(* CoDeSys 2.3.9.48 project: PLC128.pro *)
(* Libraries: WagoLibSockets.lib 14.5.12 12:49:54, SysLibSockets.lib 5.5.11 09:22:24, Standard.lib 8.11.10 12:37:48, SYSLIBCALLBACK.LIB 8.11.10 12:37:48, NETVARUDP_LIB_V23.LIB 8.11.10 12:37:48 *)

(* PLC configuration (modules and I/O channels)
IN1 AT %IX2.0 [BOOLOnX_I] Ch_1 Digital input
IN2 AT %IX2.1 [BOOLOnX_I] Ch_2 Digital input
IN3 AT %IX2.2 [BOOLOnX_I] Ch_3 Digital input
IN4 AT %IX2.3 [BOOLOnX_I] Ch_4 Digital input
IN5 AT %IX2.4 [BOOLOnX_I] Ch_5 Digital input
IN6 AT %IX2.5 [BOOLOnX_I] Ch_6 Digital input
IN7 AT %IX2.6 [BOOLOnX_I] Ch_7 Digital input
IN8 AT %IX2.7 [BOOLOnX_I] Ch_8 Digital input
0750-0530 8 DO 24 V DC 0.5A [Type_10_8_Channels] node 1, in %IB4 out %QB4 {INTTypePAAssignment = fieldbus2; INTTypeModule = plugged}
  AT %QX2.0 [BOOLOnX_Q] Ch_1 Digital output
  AT %QX2.1 [BOOLOnX_Q] Ch_2 Digital output
  AT %QX2.2 [BOOLOnX_Q] Ch_3 Digital output
  AT %QX2.3 [BOOLOnX_Q] Ch_4 Digital output
  AT %QX2.4 [BOOLOnX_Q] Ch_5 Digital output
  AT %QX2.5 [BOOLOnX_Q] Ch_6 Digital output
  AT %QX2.6 [BOOLOnX_Q] Ch_7 Digital output
  AT %QX2.7 [BOOLOnX_Q] Ch_8 Digital output
0750-0653 RS485 Interface [Type_21_1_Channels] node 2, in %IB0 out %QB0 {INTTypePAAssignment = fieldbus2; INTTypeModule = plugged}
  AT %IX0.0 [BOOLOnX_I] Transmission acknowledgement
  AT %IX0.1 [BOOLOnX_I] Reception request
  AT %IX0.2 [BOOLOnX_I] Initialization acknowledgement
  AT %IX0.3 [BOOLOnX_I] Input buffer is full
  AT %IX0.4 [BOOLOnX_I] Number of received characters Bit 0
  AT %IX0.5 [BOOLOnX_I] Number of received characters Bit 1
  AT %IX0.6 [BOOLOnX_I] Number of received characters Bit 2
  AT %IB1 [BYTEOnB_I] Input data Byte 0
  AT %IB2 [BYTEOnB_I] Input data Byte 1
  AT %IB3 [BYTEOnB_I] Input data Byte 2
  AT %QX0.0 [BOOLOnX_Q] Transmission request
  AT %QX0.1 [BOOLOnX_Q] Reception acknowledgement
  AT %QX0.2 [BOOLOnX_Q] Initialization request
  AT %QX0.4 [BOOLOnX_Q] Number of characters Bit 0
  AT %QX0.5 [BOOLOnX_Q] Number of characters Bit 1
  AT %QX0.6 [BOOLOnX_Q] Number of characters Bit 2
  AT %QB1 [BYTEOnB_Q] Output data Byte 0
  AT %QB2 [BYTEOnB_Q] Output data Byte 1
  AT %QB3 [BYTEOnB_Q] Output data Byte 2
fb_var0 AT %ID128 [DWORDOnD_I] DWORD
DWORD, Fieldbus input [FBVAR_DWORD_IN] node 2, in %IB0 out %QB0
  fb_var4 AT %ID129 [DWORDOnD_I] DWORD
DWORD, Fieldbus output [FBVAR_DWORD_OUT] node 3, in %IB0 out %QB0
  fb_var9 AT %QD128 [DWORDOnD_Q] DWORD
DWORD, Fieldbus output [FBVAR_DWORD_OUT] node 4, in %IB0 out %QB0
  fb_var8 AT %QD129 [DWORDOnD_Q] DWORD
DWORD, Fieldbus output [FBVAR_DWORD_OUT] node 5, in %IB0 out %QB0
  fb_var7 AT %QD130 [DWORDOnD_Q] DWORD
DWORD, Fieldbus output [FBVAR_DWORD_OUT] node 6, in %IB0 out %QB0
  fb_var6 AT %QD131 [DWORDOnD_Q] DWORD
DWORD, Fieldbus output [FBVAR_DWORD_OUT] node 7, in %IB0 out %QB0
  fb_var5 AT %QD132 [DWORDOnD_Q] DWORD
DWORD, Fieldbus input [FBVAR_DWORD_IN] node 8, in %IB0 out %QB0
  fb_var3 AT %ID130 [DWORDOnD_I] DWORD
DWORD, Fieldbus input [FBVAR_DWORD_IN] node 9, in %IB0 out %QB0
  fb_var2 AT %ID131 [DWORDOnD_I] DWORD
DWORD, Fieldbus input [FBVAR_DWORD_IN] node 10, in %IB0 out %QB0
  fb_var1 AT %ID132 [DWORDOnD_I] DWORD
Flag variables [FLAG_VARS] node 2, in %IB0 out %QB0
Modbus-Master [MB_MASTER] node 3, in %IB0 out %QB0
*)

(* Task configuration *)
TASK TCPServer (PRIORITY := 1, INTERVAL := T#100ms);
	TCPServer();
END_TASK

(* Global variable list: Networkmanagement implicit Variables UDP *)
VAR_GLOBAL CONSTANT
	USE_NWVARS_UDP : BOOL := FALSE;
	MAX_NetVarItems_UDP	: INT := 0;
	MAX_NetVarPDO_Rx_UDP	: INT := 0;
	MAX_NetVarPDO_Tx_UDP	: INT := 0;
	MAX_NetVarOD_UDP		: INT := 0;
END_VAR
VAR_GLOBAL
	pNetVarItems_UDP		: ARRAY[0..MAX_NetVarItems_UDP] OF NetVarDataItem_UDP;
	pNetVarPDO_Rx_UDP		: ARRAY[0..MAX_NetVarPDO_Rx_UDP] OF NetVarPDO_Rx_UDP;
	pNetVarPDO_Tx_UDP		: ARRAY[0..MAX_NetVarPDO_Tx_UDP] OF NetVarPDO_Tx_UDP;
	pNetVarOD_UDP			: ARRAY[0..MAX_NetVarOD_UDP] OF NetVarSDO_UDP;
	pNetVarPDO_Rx_Diagnosis_UDP : ARRAY[0..MAX_NetVarPDO_Rx_UDP] OF NetVarUDPDiagStruct;
	pNetVarPDO_Tx_Diagnosis_UDP : ARRAY[0..MAX_NetVarPDO_Tx_UDP] OF NetVarUDPDiagStruct;
END_VAR

(* POU TCPServer, ST *)
PROGRAM TCPServer
VAR
	diSocket : DINT := -1;
	iPort : INT:=10000;
	Client : CLIENT_ACCEPT := (diSocket := -1);

	bySend :ARRAY [0..5] OF BYTE;
	byRecv : STRING;
	ArrayRecv1 : ARRAY[0..1024] OF STRING;
	ArrayRecv2 : ARRAY[0..1024] OF STRING;
	Reply : CLIENT_REPLY;
	bCloseClient: BOOL;
	bActive: BOOL := TRUE;
	test: STRING;
	number: INT;
END_VAR
IF bActive THEN
	IF diSocket = -1 THEN
		diSocket := TcpServerOpenSocket(iPort, 10, 0);
	END_IF

	IF  Client.diSocket = -1 THEN
		Client := TcpServerWaitForConnect(diSocket, 1);
	END_IF

	IF  Client.diSocket <> -1 THEN
		(*TcpSendData(Client.diSocket, ADR(bySend), SIZEOF(bySend), 2)*);
		TcpReceiveData(Client.diSocket, ADR(byRecv), SIZEOF(byRecv), 4);
		test := MID(byRecv, 1, 4);
		number := STRING_TO_INT(test);
		ArrayRecv1[number] := byRecv;
		bCloseClient := TRUE;
	END_IF

	IF bCloseClient THEN
		bCloseClient := FALSE;
		SysSockClose(diSocket:=Client.diSocket);
		Client.diSocket := -1;
	END_IF
END_IF
END_PROGRAM

(* POU TcpServerOpenSocket, ST *)
FUNCTION TcpServerOpenSocket : DINT
VAR_INPUT
	iPort:INT;						(* Port number *)
	diMaxConnections:DINT;		(* Max possible client connections of the server *)
	diMaxDataSize:DINT;			(* Max size of data to transmitt; if size = 0 default values are used *)
END_VAR
VAR
	diSocket:DINT;
	bResult:BOOL;
	sa:SOCKADDRESS;
	bOptNoDelay:BOOL;
	lOptLinger:SOCKET_LINGER;
END_VAR
diSocket:=SysSockCreate(SOCKET_AF_INET, SOCKET_STREAM, SOCKET_IPPROTO_IP);
IF diSocket <> SOCKET_INVALID THEN
	sa.sin_family:=SOCKET_AF_INET;
	sa.sin_addr:=SOCKET_INADDR_ANY;
	sa.sin_port:=SysSockHtons(iPort);
	bResult:=SysSockBind(diSocket, ADR(sa), SIZEOF(sa));
	IF bResult = FALSE THEN
		diSocket:=SOCKET_INVALID;
	ELSE
		bResult:=SysSockListen(diSocket, diMaxConnections);
		IF bResult = FALSE THEN
			diSocket:=SOCKET_INVALID;
		END_IF
	END_IF
END_IF
TcpServerOpenSocket:=diSocket;
END_FUNCTION

(* POU TcpServerWaitForConnect, ST *)
FUNCTION TcpServerWaitForConnect : CLIENT_ACCEPT
VAR_INPUT
	diServerSocket:DINT;
	diTimeout : DINT;	(* Timeout in seconds *)
END_VAR
VAR
	sa:SOCKADDRESS;
	ia:INADDR;
	diSize:DINT;
	fdRead: SOCKET_FD_SET;
	fdWrite:SOCKET_FD_SET;
	fdExcept:SOCKET_FD_SET;
	tvTimeout:SOCKET_TIMEVAL;
END_VAR
tvTimeout.tv_sec := diTimeout ;
tvTimeout.tv_usec := 0;
fdRead.fd_count := 1;
fdRead.fd_array[0] := diServerSocket;
IF (SysSockSelect(SOCKET_FD_SETSIZE, ADR(fdRead), 0, 0, ADR(tvTimeout)) > 0) THEN
	diSize:=SIZEOF(sa);
	TcpServerWaitForConnect.diSocket:=SysSockAccept(diServerSocket, ADR(sa), ADR(diSize));
	ia.S_addr:=DINT_TO_DWORD(sa.sin_addr);
	SysSockInetNtoa(ia, TcpServerWaitForConnect.stIPAddress, SIZEOF(TcpServerWaitForConnect.stIPAddress));
ELSE
	TcpServerWaitForConnect.diSocket := -1;
END_IF
END_FUNCTION

(* POU TcpReceiveData, ST *)
FUNCTION TcpReceiveData : DINT
VAR_INPUT
	diSocket:DINT;		(* Socket Id *)
	pbyData:DWORD;		(* Address of data buffer *)
	diDataSize:DINT;		(* Size of data to send *)
	diTImeout : DINT;		(* Timeout in seconds *)
END_VAR
VAR
	fdRead:SOCKET_FD_SET;
	tvTimeout:SOCKET_TIMEVAL;
END_VAR
tvTimeout.tv_sec := diTimeout ;
tvTimeout.tv_usec := 0;
fdRead.fd_count := 1;
fdRead.fd_array[0] := diSocket;
IF (SysSockSelect(SOCKET_FD_SETSIZE, ADR(fdRead), 0, 0, ADR(tvTimeout)) > 0) THEN
	TcpReceiveData:=SysSockRecv(diSocket, pbyData, diDataSize, 0);
END_IF
END_FUNCTION

(* POU PLC_PRG, ST *)
PROGRAM PLC_PRG
VAR
END_VAR
%QX2.0 := TRUE;
END_PROGRAM

(* POU Configuration/MODBUS_CONFIGURATION, ST *)
PROGRAM MODBUS_CONFIGURATION        
VAR                                
END_VAR                            
(*                                 
   <?xml version="1.0" encoding="UTF-16" standalone="yes"?>
<network xml_structure_version="1" xml_feature_version="1">
	<generator_settings minRTUTaskCycleTimeMs="5" minEthaskCycleTimeMs="5" ethSlaveMultiplier="0.1" rtuInterfaceMultiplier="0.1" taskGeneration="true"/>
</network>
                              
*)                                 
;                                  
END_PROGRAM

(* POU TcpSendData, ST *)
FUNCTION TcpSendData : DINT
VAR_INPUT
	diSocket:DINT;		(* Socket Id *)
	pbyData:DWORD;		(* Address of data buffer *)
	diDataSize:DINT;		(* Size of data to send *)
	diTImeout : DINT;		(* Timeout in seconds *)
END_VAR
VAR
	fdWrite:SOCKET_FD_SET;
	tvTimeout:SOCKET_TIMEVAL;
END_VAR
tvTimeout.tv_sec := diTimeout ;
tvTimeout.tv_usec := 0;
fdWrite.fd_count := 1;
fdWrite.fd_array[0] := diSocket;
IF (SysSockSelect(SOCKET_FD_SETSIZE, 0, ADR(fdWrite), 0, ADR(tvTimeout)) > 0) THEN
	TcpSendData:=SysSockSend(diSocket, pbyData, diDataSize, 0);
END_IF
END_FUNCTION
